//	KPV15du	: BOOL;
END_VAR
(* global variable list tmr *)
{attribute 'qualified_only' := ''}
{attribute 'symbol' := 'none'}
VAR_GLOBAL
	///Unlock
	//Unlock: Ttonp := (pt := TIME#3s0ms);
	crsPmStarter_20	: TON := ( PT := TIME#20S0MS );	// 20	
//	crsNIgnition_10: TON := (pt := TIME#0S0MS);	// 10	
//	crsNBoost_10: TON := (pt := TIME#0S0MS);	// 10
	KPV234_wOpen	: TON := ( PT := TIME#10S0MS );	// 10
	KPV15_wOpen		: TON := ( PT := TIME#10S0MS );	// 10
	KPV15_nOpen		: TON := ( PT := TIME#10S0MS );	// 10
	// задержка выключения насосов после останова
	PNU_S_Off		: TON := ( PT := TIME#5M );	// 30 minutes // 5 minutes 14_07_2025
	// задержка отключения насосов при подкачке масла Н на этапе прогрева или охлаждения двигателя
	PNU_S_pumpH		: TOF := ( PT := TIME#1M );	// 1 minutes
END_VAR
(* global variable list acpar_handler *)
{attribute 'qualified_only' := ''}
VAR_GLOBAL
	handler: TAcparHandler;
END_VAR
(* global variable list FuelReg *)
{region INFO}
(*
Назначение: Числовые настройки
Автор     : Дергаев
Дата      : 12.05.2025 16:11:36
Версия    : 00.01.00
*)
{endregion}
{attribute 'qualified_only'}
{attribute 'symbol' := 'none'}
VAR_GLOBAL
{attribute 'symbol' := 'readwrite'}
  {attribute 'export' := '("archive":"True","communication":("cycle":"base"),"name":"Верхнее ограничение Nтк","units": "об/мин","digit": "0","limit": ("low": "0.0","high": "9000.0"))'}
  limValUpNvd  : Ttunpar := (value := REAL#8350.0, set_value := REAL#8350.0, enable_valueLimit := TRUE, lolim := REAL#0.0, hilim := REAL#9000.0, enable_direct_update := TRUE); 
{attribute 'symbol' := 'readwrite'}
  {attribute 'export' := '("archive":"True","communication":("cycle":"base"),"name":"Верхнее ограничение Nст","units": "об/мин","digit": "0","limit": ("low": "0.0","high": "9000.0"))'}
  limValUpNst  : Ttunpar := (value := REAL#8500.0, set_value := REAL#8500.0, enable_valueLimit := TRUE, lolim := REAL#0.0, hilim := REAL#9000.0, enable_direct_update := TRUE); 
{attribute 'symbol' := 'readwrite'}
  {attribute 'export' := '("archive":"True","communication":("cycle":"base"),"name":"Верхнее ограничение Тст","units": "°C","digit": "0","limit": ("low": "0.0","high": "800.0"))'}
  limValUpTst  : Ttunpar := (value := REAL#650.0, set_value := REAL#650.0, enable_valueLimit := TRUE, lolim := REAL#0.0, hilim := REAL#800.0, enable_direct_update := TRUE); 
{attribute 'symbol' := 'readwrite'}
  {attribute 'export' := '("archive":"True","communication":("cycle":"base"),"name":"Верх. огр. Тст на пуске","units": "°С","digit": "0","limit": ("low": "0.0","high": "800.0"))'}
  limValUpTstStart : Ttunpar := (value := REAL#680.0, set_value := REAL#680.0, enable_valueLimit := TRUE, lolim := REAL#0.0, hilim := REAL#800.0, enable_direct_update := TRUE); 
{attribute 'symbol' := 'readwrite'}
  {attribute 'export' := '("archive":"True","communication":("cycle":"base"),"name":"Верхнее ограничение Рк","units": "МПа","digit": "2","limit": ("low": "0.0","high": "2.0"))'}
  limValUpPk  : Ttunpar := (value := REAL#1.4, set_value := REAL#1.4, enable_valueLimit := TRUE, lolim := REAL#0.0, hilim := REAL#2.0, enable_direct_update := TRUE); 
{attribute 'symbol' := 'readwrite'}
  {attribute 'export' := '("archive":"True","communication":("cycle":"base"),"name":"Рег. Верхнее ограничение Nтк","units": "об/мин","digit": "0","limit": ("low": "-500.0","high": "500.0"))'}
  RegLimValUpNvd  : Ttunpar := (value := REAL#0.0, set_value := REAL#0.0, enable_valueLimit := TRUE, lolim := REAL#-500.0, hilim := REAL#500.0, enable_direct_update := TRUE); 
{attribute 'symbol' := 'readwrite'}
  {attribute 'export' := '("archive":"True","communication":("cycle":"base"),"name":"Рег. Нижнее ограничение Nтк","units": "об/мин","digit": "0","limit": ("low": "-500.0","high": "500.0"))'}
  RegLimValDnNvd  : Ttunpar := (value := REAL#300.0, set_value := REAL#300.0, enable_valueLimit := TRUE, lolim := REAL#-500.0, hilim := REAL#500.0, enable_direct_update := TRUE); 
{attribute 'symbol' := 'readwrite'}
  {attribute 'export' := '("archive":"True","communication":("cycle":"base"),"name":"Рег. Верхнее ограничение Nст","units": "об/мин","digit": "0","limit": ("low": "-500.0","high": "500.0"))'}
  RegLimValUpNst  : Ttunpar := (value := REAL#0.0, set_value := REAL#0.0, enable_valueLimit := TRUE, lolim := REAL#-500.0, hilim := REAL#500.0, enable_direct_update := TRUE); 
{attribute 'symbol' := 'readwrite'}
  {attribute 'export' := '("archive":"True","communication":("cycle":"base"),"name":"Рег. Верхнее ограничение Тст","units": "°C","digit": "0","limit": ("low": "-200.0","high": "200.0"))'}
  RegLimValUpTst  : Ttunpar := (value := REAL#0.0, set_value := REAL#0.0, enable_valueLimit := TRUE, lolim := REAL#-200.0, hilim := REAL#200.0, enable_direct_update := TRUE); 
{attribute 'symbol' := 'readwrite'}
  {attribute 'export' := '("archive":"True","communication":("cycle":"base"),"name":"Рег. Верх. огр. Тст на пуске","units": "°С","digit": "0","limit": ("low": "-200.0","high": "200.0"))'}
  RegLimValUpTstStart : Ttunpar := (value := REAL#0.0, set_value := REAL#0.0, enable_valueLimit := TRUE, lolim := REAL#-200.0, hilim := REAL#200.0, enable_direct_update := TRUE); 
{attribute 'symbol' := 'readwrite'}
  {attribute 'export' := '("archive":"True","communication":("cycle":"base"),"name":"Рег. Верхнее ограничение Рк","units": "МПа","digit": "2","limit": ("low": "-0.5","high": "0.5"))'}
  RegLimValUpPk  : Ttunpar := (value := REAL#0.0, set_value := REAL#0.0, enable_valueLimit := TRUE, lolim := REAL#-0.5, hilim := REAL#0.5, enable_direct_update := TRUE); 
{attribute 'symbol' := 'readwrite'}
  {attribute 'export' := '("archive":"True","communication":("cycle":"base"),"name":"Ступенька на розжиг ","units": "кг/ч","digit": "0","limit": ("low": "0.0","high": "1000.0"))'}
  ignitionStep  : Ttunpar := (value := REAL#100.0, set_value := REAL#100.0, enable_valueLimit := TRUE, lolim := REAL#0.0, hilim := REAL#1000.0, enable_direct_update := TRUE); 
{attribute 'symbol' := 'readwrite'}
  {attribute 'export' := '("archive":"True","communication":("cycle":"base"),"name":"Пауза на первой ступеньке ","units": "с","digit": "0","limit": ("low": "0.0","high": "60.0"))'}
  ignitionDelay  : Ttunpar := (value := REAL#3.0, set_value := REAL#3.0, enable_valueLimit := TRUE, lolim := REAL#0.0, hilim := REAL#60.0, enable_direct_update := TRUE); 
{attribute 'symbol' := 'readwrite'}
  {attribute 'export' := '("archive":"True","communication":("cycle":"base"),"name":"Макс. длительность розжига ","units": "с","digit": "0","limit": ("low": "0.0","high": "60.0"))'}
  ignitionMaxTime  : Ttunpar := (value := REAL#10.0, set_value := REAL#10.0, enable_valueLimit := TRUE, lolim := REAL#0.0, hilim := REAL#60.0, enable_direct_update := TRUE); 
{attribute 'symbol' := 'readwrite'}
  {attribute 'export' := '("archive":"True","communication":("cycle":"base"),"name":"Макс. Gт на розжиге","units": "кг/ч","digit": "0","limit": ("low": "0.0","high": "1000.0"))'}
  ignitionMaxVal  : Ttunpar := (value := REAL#250.0, set_value := REAL#250.0, enable_valueLimit := TRUE, lolim := REAL#0.0, hilim := REAL#1000.0, enable_direct_update := TRUE); 
{attribute 'symbol' := 'readwrite'}
  {attribute 'export' := '("archive":"True","communication":("cycle":"base"),"name":"Темп программного разгона","units": "[кг/ч]/c","digit": "0","limit": ("low": "0.0","high": "1000.0"))'}
  rateOnProg  : Ttunpar := (value := REAL#30.0, set_value := REAL#30.0, enable_valueLimit := TRUE, lolim := REAL#0.0, hilim := REAL#1000.0, enable_direct_update := TRUE); 
{attribute 'symbol' := 'readwrite'}
  {attribute 'export' := '("archive":"True","communication":("cycle":"base"),"name":"Ступенька при прог. разгоне ","units": "кг/ч","digit": "0","limit": ("low": "0.0","high": "1000.0"))'}
  stepOnProg  : Ttunpar := (value := REAL#0.0, set_value := REAL#0.0, enable_valueLimit := TRUE, lolim := REAL#0.0, hilim := REAL#1000.0, enable_direct_update := TRUE); 
{attribute 'symbol' := 'readwrite'}
  {attribute 'export' := '("archive":"True","communication":("cycle":"base"),"name":"T1 регулирования Nтк","units": "с","digit": "2","limit": ("low": "0.0","high": "10.0"))'}
  tau1vd  : Ttunpar := (value := REAL#0.5, set_value := REAL#0.5, enable_valueLimit := TRUE, lolim := REAL#0.0, hilim := REAL#10.0, enable_direct_update := TRUE); 
{attribute 'symbol' := 'readwrite'}
  {attribute 'export' := '("archive":"True","communication":("cycle":"base"),"name":"T2 регулирования Nтк","units": "с","digit": "2","limit": ("low": "0.0","high": "10.0"))'}
  tau2vd  : Ttunpar := (value := REAL#0.1, set_value := REAL#0.1, enable_valueLimit := TRUE, lolim := REAL#0.0, hilim := REAL#10.0, enable_direct_update := TRUE); 
{attribute 'symbol' := 'readwrite'}
  {attribute 'export' := '("archive":"True","communication":("cycle":"base"),"name":"T1 регулирования Nст","units": "с","digit": "2","limit": ("low": "0.0","high": "10.0"))'}
  tau1st  : Ttunpar := (value := REAL#0.5, set_value := REAL#0.5, enable_valueLimit := TRUE, lolim := REAL#0.0, hilim := REAL#10.0, enable_direct_update := TRUE); 
{attribute 'symbol' := 'readwrite'}
  {attribute 'export' := '("archive":"True","communication":("cycle":"base"),"name":"Т2 регулирования Nст","units": "с","digit": "2","limit": ("low": "0.0","high": "10.0"))'}
  tau2st : Ttunpar := (value := REAL#0.1, set_value := REAL#0.1, enable_valueLimit := TRUE, lolim := REAL#0.0, hilim := REAL#10.0, enable_direct_update := TRUE); 
{attribute 'symbol' := 'readwrite'}
  {attribute 'export' := '("archive":"True","communication":("cycle":"base"),"name":"Т1 регулирования Тст","units": "с","digit": "2","limit": ("low": "0.0","high": "10.0"))'}
  tau1Tst  : Ttunpar := (value := REAL#0.5, set_value := REAL#0.5, enable_valueLimit := TRUE, lolim := REAL#0.0, hilim := REAL#10.0, enable_direct_update := TRUE); 
{attribute 'symbol' := 'readwrite'}
  {attribute 'export' := '("archive":"True","communication":("cycle":"base"),"name":"Т2 регулирования Тст","units": "с","digit": "2","limit": ("low": "0.0","high": "10.0"))'}
  tau2Tst  : Ttunpar := (value := REAL#0.1, set_value := REAL#0.1, enable_valueLimit := TRUE, lolim := REAL#0.0, hilim := REAL#10.0, enable_direct_update := TRUE); 
{attribute 'symbol' := 'readwrite'}
  {attribute 'export' := '("archive":"True","communication":("cycle":"base"),"name":"Т1 регулирования Рк","units": "с","digit": "2","limit": ("low": "0.0","high": "10.0"))'}
  tau1Pk  : Ttunpar := (value := REAL#0.5, set_value := REAL#0.5, enable_valueLimit := TRUE, lolim := REAL#0.0, hilim := REAL#10.0, enable_direct_update := TRUE); 
{attribute 'symbol' := 'readwrite'}
  {attribute 'export' := '("archive":"True","communication":("cycle":"base"),"name":"Т2 регулирования Рк","units": "с","digit": "2","limit": ("low": "0.0","high": "10.0"))'}
  tau2Pk  : Ttunpar := (value := REAL#0.1, set_value := REAL#0.1, enable_valueLimit := TRUE, lolim := REAL#0.0, hilim := REAL#10.0, enable_direct_update := TRUE); 
{attribute 'symbol' := 'readwrite'}
  {attribute 'export' := '("archive":"True","communication":("cycle":"base"),"name":"DZ регулирования Nтк","units": "об/мин","digit": "1","limit": ("low": "0.0","high": "100.0"))'}
  dzVd  : Ttunpar := (value := REAL#2.0, set_value := REAL#2.0, enable_valueLimit := TRUE, lolim := REAL#0.0, hilim := REAL#100.0, enable_direct_update := TRUE); 
{attribute 'symbol' := 'readwrite'}
  {attribute 'export' := '("archive":"True","communication":("cycle":"base"),"name":"DZ регулирования Nст","units": "об/мин","digit": "1","limit": ("low": "0.0","high": "100.0"))'}
  dzSt  : Ttunpar := (value := REAL#2.0, set_value := REAL#2.0, enable_valueLimit := TRUE, lolim := REAL#0.0, hilim := REAL#100.0, enable_direct_update := TRUE); 
{attribute 'symbol' := 'readwrite'}
  {attribute 'export' := '("archive":"True","communication":("cycle":"base"),"name":"DZ регулирования Тст","units": "°С","digit": "1","limit": ("low": "0.0","high": "100.0"))'}
  dzTst  : Ttunpar := (value := REAL#1.0, set_value := REAL#1.0, enable_valueLimit := TRUE, lolim := REAL#0.0, hilim := REAL#100.0, enable_direct_update := TRUE); 
{attribute 'symbol' := 'readwrite'}
  {attribute 'export' := '("archive":"True","communication":("cycle":"base"),"name":"DZ регулирования Рк","units": "МПа","digit": "2","limit": ("low": "0.0","high": "0.2"))'}
  dzPk  : Ttunpar := (value := REAL#0.01, set_value := REAL#0.01, enable_valueLimit := TRUE, lolim := REAL#0.0, hilim := REAL#0.2, enable_direct_update := TRUE); 
{attribute 'symbol' := 'readwrite'}
  {attribute 'export' := '("archive":"True","communication":("cycle":"base"),"name":"К рабочего регулятора Nтк","units": "","digit": "2","limit": ("low": "0.0","high": "50.0"))'}
  kRVd  : Ttunpar := (value := REAL#0.0001, set_value := REAL#0.0001, enable_valueLimit := TRUE, lolim := REAL#0.0, hilim := REAL#50.0, enable_direct_update := TRUE); 
{attribute 'symbol' := 'readwrite'}
  {attribute 'export' := '("archive":"True","communication":("cycle":"base"),"name":"К верхнего ограничителя Nтк","units": "","digit": "2","limit": ("low": "0.0","high": "50.0"))'}
  kLupVd  : Ttunpar := (value := REAL#0.1, set_value := REAL#0.1, enable_valueLimit := TRUE, lolim := REAL#0.0, hilim := REAL#50.0, enable_direct_update := TRUE); 
{attribute 'symbol' := 'readwrite'}
  {attribute 'export' := '("archive":"True","communication":("cycle":"base"),"name":"К нижнего ограничителя Nтк","units": "","digit": "2","limit": ("low": "0.0","high": "50.0"))'}
  kLdnVd  : Ttunpar := (value := REAL#0.1, set_value := REAL#0.1, enable_valueLimit := TRUE, lolim := REAL#0.0, hilim := REAL#50.0, enable_direct_update := TRUE); 
{attribute 'symbol' := 'readwrite'}
  {attribute 'export' := '("archive":"True","communication":("cycle":"base"),"name":"К рабочего регулятора Nст","units": "","digit": "2","limit": ("low": "0.0","high": "50.0"))'}
  kRst  : Ttunpar := (value := REAL#0.0001, set_value := REAL#0.0001, enable_valueLimit := TRUE, lolim := REAL#0.0, hilim := REAL#50.0, enable_direct_update := TRUE); 
{attribute 'symbol' := 'readwrite'}
  {attribute 'export' := '("archive":"True","communication":("cycle":"base"),"name":"К верхнего ограничителя Nст","units": "","digit": "2","limit": ("low": "0.0","high": "50.0"))'}
  kLupST  : Ttunpar := (value := REAL#0.1, set_value := REAL#0.1, enable_valueLimit := TRUE, lolim := REAL#0.0, hilim := REAL#50.0, enable_direct_update := TRUE); 
{attribute 'symbol' := 'readwrite'}
  {attribute 'export' := '("archive":"True","communication":("cycle":"base"),"name":"К верхнего ограничителя Тст","units": "","digit": "2","limit": ("low": "0.0","high": "50.0"))'}
  kLupTst  : Ttunpar := (value := REAL#0.1, set_value := REAL#0.1, enable_valueLimit := TRUE, lolim := REAL#0.0, hilim := REAL#50.0, enable_direct_update := TRUE); 
{attribute 'symbol' := 'readwrite'}
  {attribute 'export' := '("archive":"True","communication":("cycle":"base"),"name":"К верхнего ограничителя Рк","units": "","digit": "2","limit": ("low": "0.0","high": "50.0"))'}
  kLupPk  : Ttunpar := (value := REAL#0.1, set_value := REAL#0.1, enable_valueLimit := TRUE, lolim := REAL#0.0, hilim := REAL#50.0, enable_direct_update := TRUE); 
{attribute 'symbol' := 'readwrite'}
  {attribute 'export' := '("archive":"True","communication":("cycle":"base"),"name":"К коррекции Nтк","units": "[об/мин]/[кг/ч]","digit": "4","limit": ("low": "0.0","high": "50.0"))'}
   kCorrNvd : Ttunpar := (value := REAL#4.0, set_value := REAL#4.0, enable_valueLimit := TRUE, lolim := REAL#0.0, hilim := REAL#50.0, enable_direct_update := TRUE); 
{attribute 'symbol' := 'readwrite'}
  {attribute 'export' := '("archive":"True","communication":("cycle":"base"),"name":"К коррекции Nст","units": "[об/мин]/[кг/ч]","digit": "4","limit": ("low": "0.0","high": "50.0"))'}
   kCorrNst : Ttunpar := (value := REAL#4.0, set_value := REAL#4.0, enable_valueLimit := TRUE, lolim := REAL#0.0, hilim := REAL#50.0, enable_direct_update := TRUE); 
{attribute 'symbol' := 'readwrite'}
  {attribute 'export' := '("archive":"True","communication":("cycle":"base"),"name":"К коррекции Tст","units": "°С/[кг/ч]","digit": "1","limit": ("low": "0.0","high": "50.0"))'}
   kCorrTst : Ttunpar := (value := REAL#0.3, set_value := REAL#0.3, enable_valueLimit := TRUE, lolim := REAL#0.0, hilim := REAL#50.0, enable_direct_update := TRUE); 
{attribute 'symbol' := 'readwrite'}
  {attribute 'export' := '("archive":"True","communication":("cycle":"base"),"name":"К коррекции Рк","units": "МПа/[кг/ч]","digit": "1","limit": ("low": "0.0","high": "50.0"))'}
   kCorrPk  : Ttunpar := (value := REAL#0.0005, set_value := REAL#0.0005, enable_valueLimit := TRUE, lolim := REAL#0.0, hilim := REAL#50.0, enable_direct_update := TRUE); 
{attribute 'symbol' := 'readwrite'}
  {attribute 'export' := '("archive":"True","communication":("cycle":"base"),"name":"Обороты вкл. рег. по Nтк","units": "об/мин","digit": "0","limit": ("low": "0.0","high": "8000.0"))'}
  setNvdRegOn  : Ttunpar := (value := REAL#6300.0, set_value := REAL#6300.0, enable_valueLimit := TRUE, lolim := REAL#0.0, hilim := REAL#8000.0, enable_direct_update := TRUE); 
{attribute 'symbol' := 'readwrite'}
  {attribute 'export' := '("archive":"True","communication":("cycle":"base"),"name":"Обороты выключения стартера","units": "об/мин","digit": "0","limit": ("low": "0.0","high": "8000.0"))'}
  setNvdStarterOff  : Ttunpar := (value := REAL#4500.0, set_value := REAL#4500.0, enable_valueLimit := TRUE, lolim := REAL#0.0, hilim := REAL#8000.0, enable_direct_update := TRUE); 
{attribute 'symbol' := 'readwrite'}
  {attribute 'export' := '("archive":"True","communication":("cycle":"base"),"name":"Обороты прогрева","units": "об/мин","digit": "0","limit": ("low": "0.0","high": "8000.0"))'}
  setNvdHeat  : Ttunpar := (value := REAL#6800.0, set_value := REAL#6800.0, enable_valueLimit := TRUE, lolim := REAL#0.0, hilim := REAL#8000.0, enable_direct_update := TRUE); 
{attribute 'symbol' := 'readwrite'}
  {attribute 'export' := '("archive":"True","communication":("cycle":"base"),"name":"Время прогрева","units": "с","digit": "0","limit": ("low": "0.0","high": "500.0"))'}
  setHeatTime  : Ttunpar := (value := REAL#300.0, set_value := REAL#300.0, enable_valueLimit := TRUE, lolim := REAL#0.0, hilim := REAL#500.0, enable_direct_update := TRUE); 
{attribute 'symbol' := 'readwrite'}
  {attribute 'export' := '("archive":"True","communication":("cycle":"base"),"name":"Обороты охлаждения","units": "об/мин","digit": "0","limit": ("low": "0.0","high": "8000.0"))'}
  setNvdCool  : Ttunpar := (value := REAL#6700.0, set_value := REAL#6700.0, enable_valueLimit := TRUE, lolim := REAL#0.0, hilim := REAL#8000.0, enable_direct_update := TRUE); 
{attribute 'symbol' := 'readwrite'}
  {attribute 'export' := '("archive":"True","communication":("cycle":"base"),"name":"Время охлаждения","units": "с","digit": "0","limit": ("low": "0.0","high": "500.0"))'}
  setCoolTime  : Ttunpar := (value := REAL#300.0, set_value := REAL#300.0, enable_valueLimit := TRUE, lolim := REAL#0.0, hilim := REAL#500.0, enable_direct_update := TRUE); 
{attribute 'symbol' := 'readwrite'}
  {attribute 'export' := '("archive":"True","communication":("cycle":"base"),"name":"Ступенька Т на пуске","units": "°С","digit": "0","limit": ("low": "0.0","high": "500.0"))'}
  setDTign  : Ttunpar := (value := REAL#100.0, set_value := REAL#100.0, enable_valueLimit := TRUE, lolim := REAL#0.0, hilim := REAL#500.0, enable_direct_update := TRUE); 
{attribute 'symbol' := 'readwrite'}
  {attribute 'export' := '("archive":"True","communication":("cycle":"base"),"name":"dNтк до верх. границы - сигн.","units": "об/мин","digit": "0","limit": ("low": "0.0","high": "100.0"))'}
  dNvdUpLim : Ttunpar := (value := REAL#20.0, set_value := REAL#20.0, enable_valueLimit := TRUE, lolim := REAL#0.0, hilim := REAL#100.0, enable_direct_update := TRUE); 
{attribute 'symbol' := 'readwrite'}
  {attribute 'export' := '("archive":"True","communication":("cycle":"base"),"name":"dNтк до нижн. границы - сигн.","units": "об/мин","digit": "0","limit": ("low": "0.0","high": "100.0"))'}
  dNvdDnLim : Ttunpar := (value := REAL#20.0, set_value := REAL#20.0, enable_valueLimit := TRUE, lolim := REAL#0.0, hilim := REAL#100.0, enable_direct_update := TRUE); 
{attribute 'symbol' := 'readwrite'}
  {attribute 'export' := '("archive":"True","communication":("cycle":"base"),"name":"dNст до верх. границы - сигн.","units": "об/мин","digit": "0","limit": ("low": "0.0","high": "100.0"))'}
  dNstUpLim : Ttunpar := (value := REAL#20.0, set_value := REAL#20.0, enable_valueLimit := TRUE, lolim := REAL#0.0, hilim := REAL#100.0, enable_direct_update := TRUE); 
{attribute 'symbol' := 'readwrite'}
  {attribute 'export' := '("archive":"True","communication":("cycle":"base"),"name":"dТст до верх. границы - сигн.","units": "°С","digit": "0","limit": ("low": "0.0","high": "100.0"))'}
  dTstUpLim : Ttunpar := (value := REAL#10.0, set_value := REAL#10.0, enable_valueLimit := TRUE, lolim := REAL#0.0, hilim := REAL#100.0, enable_direct_update := TRUE); 
{attribute 'symbol' := 'readwrite'}
  {attribute 'export' := '("archive":"True","communication":("cycle":"base"),"name":"dPk до верх. границы - сигн.","units": "МПа","digit": "2","limit": ("low": "0.0","high": "0.5"))'}
  dPkUpLim : Ttunpar := (value := REAL#0.1, set_value := REAL#0.1, enable_valueLimit := TRUE, lolim := REAL#0.0, hilim := REAL#0.5, enable_direct_update := TRUE); 
{attribute 'symbol' := 'readwrite'}
  {attribute 'export' := '("archive":"True","communication":("cycle":"base"),"name":"Мин. Т при работе - горение","units": "°С","digit": "0","limit": ("low": "0.0","high": "700.0"))'}
  lowTonWork : Ttunpar := (value := REAL#250.0, set_value := REAL#250.0, enable_valueLimit := TRUE, lolim := REAL#0.0, hilim := REAL#700.0, enable_direct_update := TRUE); 
{attribute 'symbol' := 'readwrite'}
  {attribute 'export' := '("archive":"True","communication":("cycle":"base"),"name":"Задержка контроля Мин.Т","units": "с","digit": "0","limit": ("low": "0.0","high": "100.0"))'}
  delayLowTonWork : Ttunpar := (value := REAL#10.0, set_value := REAL#10.0, enable_valueLimit := TRUE, lolim := REAL#0.0, hilim := REAL#100.0, enable_direct_update := TRUE); 
{attribute 'symbol' := 'readwrite'}
  {attribute 'export' := '("archive":"True","communication":("cycle":"base"),"name":"Темп разгона на регуляторе","units": "(об/мин)/c","digit": "0","limit": ("low": "0.0","high": "200.0"))'}
  rateOnReg  : Ttunpar := (value := REAL#50.0, set_value := REAL#50.0, enable_valueLimit := TRUE, lolim := REAL#0.0, hilim := REAL#200.0, enable_direct_update := TRUE); 
  // Обратная зависимость расхода топлива от степени открытия топливного клапана
  gTtoDoz : Tlinear :=
  (
    nPoint :=  17,
    point :=
    [
      (x := REAL#0.0, y := REAL#0.0),
      (x := REAL#117.0, y := REAL#6.25),
      (x := REAL#330.0, y := REAL#12.5),
      (x := REAL#555.0, y := REAL#18.75),
      (x := REAL#757.0, y := REAL#25.0),
      (x := REAL#995.0, y := REAL#31.25),
      (x := REAL#1250.0, y := REAL#37.5),
      (x := REAL#1522.0, y := REAL#43.75),
      (x := REAL#1806.0, y := REAL#50.0),
      (x := REAL#2107.0, y := REAL#56.25),
      (x := REAL#2430.0, y := REAL#62.5),
      (x := REAL#2772.0, y := REAL#68.75),
      (x := REAL#3135.0, y := REAL#75.0),
      (x := REAL#3527.0, y := REAL#81.25),
      (x := REAL#3948.0, y := REAL#87.5),
      (x := REAL#4412.0, y := REAL#93.75),
      (x := REAL#4920.0, y := REAL#100.0)
    ]
  );

  {attribute 'symbol' := 'read'}
  fReg : TRegNK12ST;
END_VAR
(* global variable list PRU *)
{attribute 'symbol' := 'read'}
{attribute 'qualified_only' := ''}
VAR_GLOBAL
	/// связь с ПРУ
	/// FALSE - отсутствие связи
	Link: BOOL;
END_VAR
(* global variable list AVOM *)
{attribute 'qualified_only' := ''}
VAR_GLOBAL
	AVOM: TAVOM;
END_VAR
(* global variable list lmt *)
{region INFO}
(*
 Назначение: Признаки срабатывания ограничительных сигнализаций
 Автор:  /Andrey/ 24.06.2025 16:50:31
 Версия: v00.00.22
 Проект: KA107__GPA2
*)
{endregion}
{attribute 'qualified_only'}
{attribute 'symbol' := 'read'}
VAR_GLOBAL
	{attribute 'symbol' := 'none'}
	common : Talarm; //Общий сигнал для VAR_STAT

END_VAR
(* global variable list BZA *)
{attribute 'symbol' := 'none'}
VAR_GLOBAL CONSTANT
	/// Уставка + доп. коэффициент
	Nst_SetUp: REAL := 3500;//2000;
	/// Уставка + доп. коэффициент
	Ntk_SetUp: REAL := 6000;//2000;
END_VAR
(* global variable list ACS *)
{attribute 'qualified_only'}
VAR_GLOBAL
	ACS			: TAutoCheckShield;
	startACS	: BOOL;		// Пуск проверки
END_VAR
(* global variable list IEC104 *)
{region INFO}
(*
 Назначение: Используется для объявления переменных, предназначенных для передачи по МЭК-104
 Автор:      /Andrey/ 16.07.2025 17:15:07
*)
{endregion}
{attribute 'qualified_only'}
{attribute 'symbol' := 'none'}
VAR_GLOBAL
	{attribute 'export' := 'an:[GVL.mde_hmi] af:[.number]'}
	GVL_mde_hmi_number : PsIEC60870.m_it_tb_1_fb; //Режим/Тип:int4/Адрес:1
	{attribute 'export' := 'an:[test.Saw_Slow] af:[.value]'}
	test_Saw_Slow_value : PsIEC60870.m_me_tf_1_fb; //Тест: пила, базовый цикл/Тип:REAL/Адрес:2
	{attribute 'export' := 'an:[test.Saw_Fast] af:[.value]'}
	test_Saw_Fast_value : PsIEC60870.m_me_tf_1_fb; //Тест: пила, быстрый цикл/Тип:REAL/Адрес:3
	{attribute 'export' := 'an:[test.Sin_Slow] af:[.value]'}
	test_Sin_Slow_value : PsIEC60870.m_me_tf_1_fb; //Тест: синус, базовый цикл/Тип:REAL/Адрес:4
	{attribute 'export' := 'an:[aipar.NTK_1] af:[.in_value]'}
	aipar_NTK_1_in_value : PsIEC60870.m_me_tf_1_fb; //Частота вращения ротора ТК (1)/Тип:REAL/Адрес:5
	{attribute 'export' := 'an:[aipar.NTK_2] af:[.in_value]'}
	aipar_NTK_2_in_value : PsIEC60870.m_me_tf_1_fb; //Частота вращения ротора ТК (2)/Тип:REAL/Адрес:6
	{attribute 'export' := 'an:[aipar.NST_1] af:[.in_value]'}
	aipar_NST_1_in_value : PsIEC60870.m_me_tf_1_fb; //Частота вращения ротора СТ (1)/Тип:REAL/Адрес:7
	{attribute 'export' := 'an:[aipar.NST_2] af:[.in_value]'}
	aipar_NST_2_in_value : PsIEC60870.m_me_tf_1_fb; //Частота вращения ротора СТ (2)/Тип:REAL/Адрес:8
	{attribute 'export' := 'an:[aipar.DG_Pos] af:[.in_value]'}
	aipar_DG_Pos_in_value : PsIEC60870.m_me_tf_1_fb; //Положение дозирующей иглы ДУС/Тип:REAL/Адрес:9
	{attribute 'export' := 'an:[aipar.Pa_out14] af:[.in_value]'}
	aipar_Pa_out14_in_value : PsIEC60870.m_me_tf_1_fb; //Давление воздуха за 14-й ступенью осевого компрессора/Тип:REAL/Адрес:10
	{attribute 'export' := 'an:[aipar.dP_conf] af:[.in_value]'}
	aipar_dP_conf_in_value : PsIEC60870.m_me_tf_1_fb; //dP на конфузоре/Тип:REAL/Адрес:11
	{attribute 'export' := 'an:[aopar.DG_Set] af:[.value]'}
	aopar_DG_Set_value : PsIEC60870.m_me_tf_1_fb; //Управление ТРК/Тип:REAL/Адрес:12
	{attribute 'export' := 'an:[dipar.SK_off] af:[.status]'}
	dipar_SK_off_status : PsIEC60870.m_bo_tb_1_fb; //СК закрыт/Тип:uint4/Адрес:13
	{attribute 'export' := 'an:[dopar.SK_ON] af:[.status]'}
	dopar_SK_ON_status : PsIEC60870.m_bo_tb_1_fb; //Открыть СК/Тип:uint4/Адрес:14
	{attribute 'export' := 'an:[aipar.DG_Pos_diag] af:[.in_value]'}
	aipar_DG_Pos_diag_in_value : PsIEC60870.m_me_tf_1_fb; //диаг. (Сигнал управления положением дозатора газа)/Тип:REAL/Адрес:15
	{attribute 'export' := 'an:[dopar.KPV15_ON] af:[.status]'}
	dopar_KPV15_ON_status : PsIEC60870.m_bo_tb_1_fb; //Открыть КПВ1, 5/Тип:uint4/Адрес:16
END_VAR
(* global variable list test *)
{attribute 'qualified_only'}
VAR_GLOBAL
	Saw_Slow	: TATestpar := ( sin_on := FALSE );
	Saw_Fast	: TATestpar := ( sin_on := FALSE );
	Sin_Slow	: TATestpar;
END_VAR
(* global variable list s_tunpar *)
{region INFO}
(*
Назначение: Числовые настройки
Автор     : Дергаев
Дата      : 20.03.2025 16:19:20
Версия    : 00.00.02
*)
{endregion}
{attribute 'qualified_only'}
{attribute 'symbol' := 'readwrite'}
VAR_GLOBAL
  {attribute 'symbol' := 'none'}
  {attribute 'export' := 'a n:[Задержка на снятие сигнала "Предпомпажное состояние"] u:[с] d:[1] lolim:[0] hilim:[1000]'}
  SAoffDelay : Ttunpar := (value := REAL#0.5, set_value := REAL#0.5, enable_direct_update := TRUE); 
  {attribute 'symbol' := 'none'}
  {attribute 'export' := 'a n:[Задержка на открытие АПРК при срабатывании сигнализатора помпажа] u:[с] d:[1] lolim:[0] hilim:[1000]'}
  SAopenDelay : Ttunpar := (value := REAL#0.0, set_value := REAL#0.0, enable_direct_update := TRUE); 
  {attribute 'symbol' := 'none'}
  {attribute 'export' := 'a n:[Задержка срабатывания сигнализатора помпажа] u:[с] d:[1] lolim:[0] hilim:[1000]'}
  SAdelay : Ttunpar := (value := REAL#2.0, set_value := REAL#2.0, enable_direct_update := TRUE); 
  {attribute 'symbol' := 'none'}
  {attribute 'export' := 'a n:[Задержка на блокировку подсчета числа срабатываний диагностики предпомпажного состояния] u:[с] d:[1] lolim:[0] hilim:[1000]'}
  blockDelay : Ttunpar := (value := REAL#2.0, set_value := REAL#2.0, enable_direct_update := TRUE); 
  {attribute 'symbol' := 'none'}
  {attribute 'export' := 'a n:[Задержка на сброс счетчика числа срабатываний диагностики предпомпажного состояния] u:[с] d:[1] lolim:[0] hilim:[1000]'}
  resetDelay : Ttunpar := (value := REAL#10.0, set_value := REAL#10.0, enable_direct_update := TRUE); 
  {attribute 'export' := 'a n:[Коэфф. при 2-й степ. осн. системы координат] u:[] d:[4] lolim:[-100] hilim:[100]'}
  c2Main : Ttunpar := (value := REAL#-0.4951, set_value := REAL#-0.4951, enable_direct_update := TRUE); 
  {attribute 'export' := 'a n:[Коэфф. при 1-й степ. осн. системы координат] u:[] d:[4] lolim:[-100] hilim:[100]'}
  c1Main : Ttunpar := (value := REAL#1.032, set_value := REAL#1.032, enable_direct_update := TRUE); 
  {attribute 'export' := 'a n:[Коэфф. при 0-й степ. осн. системы координат] u:[] d:[4] lolim:[-100] hilim:[100]'}
  c0Main : Ttunpar := (value := REAL#1.7225, set_value := REAL#1.7225, enable_direct_update := TRUE); 
  {attribute 'export' := 'a n:[Коэфф. при 2-й степ. 1-й рез. системы координат] u:[] d:[4] lolim:[-100] hilim:[100]'}
  c2Res1 : Ttunpar := (value := REAL#-0.3076, set_value := REAL#-0.3076, enable_direct_update := TRUE); 
  {attribute 'export' := 'a n:[Коэфф. при 1-й степ. 1-й рез. системы координат] u:[] d:[4] lolim:[-100] hilim:[100]'}
  c1Res1 : Ttunpar := (value := REAL#1.0322, set_value := REAL#1.0322, enable_direct_update := TRUE); 
  {attribute 'export' := 'a n:[Коэфф. при 0-й степ. 1-й рез. системы координат] u:[] d:[4] lolim:[-100] hilim:[100]'}
  c0Res1 : Ttunpar := (value := REAL#1.4, set_value := REAL#1.4, enable_direct_update := TRUE); 
  {attribute 'export' := 'a n:[Коэфф. при 2-й степ. 2-й рез. системы координат] u:[] d:[4] lolim:[-100] hilim:[100]'}
  c2Res2 : Ttunpar := (value := REAL#1.5895, set_value := REAL#1.5895, enable_direct_update := TRUE); 
  {attribute 'export' := 'a n:[Коэфф. при 1-й степ. 2-й рез. системы координат] u:[] d:[4] lolim:[-100] hilim:[100]'}
  c1Res2 : Ttunpar := (value := REAL#-1.7931, set_value := REAL#-1.7931, enable_direct_update := TRUE); 
  {attribute 'export' := 'a n:[Коэфф. при 0-й степ. 2-й рез. системы координат] u:[] d:[4] lolim:[-100] hilim:[100]'}
  c0Res2 : Ttunpar := (value := REAL#1.7433, set_value := REAL#1.7433, enable_direct_update := TRUE); 
  {attribute 'export' := 'a n:[Мин. помпажный запас] u:[%] d:[1] lolim:[0] hilim:[100]'}
  minSR : Ttunpar := (value := REAL#10.0, set_value := REAL#10.0, enable_direct_update := TRUE); 
  {attribute 'export' := 'a n:[Макс. давление на выходе Н] u:[МПа] d:[2] lolim:[0] hilim:[32]'}
  maxPout  : Ttunpar := (value := REAL#7.5, set_value := REAL#7.5, enable_direct_update := TRUE); 
  {attribute 'export' := 'a n:[Макс. степень сжатия] u:[] d:[2] lolim:[0] hilim:[3]'}
  maxPR  : Ttunpar := (value := REAL#1.27, set_value := REAL#1.27, enable_direct_update := TRUE); 
  {attribute 'export' := 'a n:[Коэффициент конфузора] u:[] d:[2] lolim:[0] hilim:[1000]'}
  Kconf : Ttunpar := (value := REAL#44.18806572, set_value := REAL#44.18806572, enable_direct_update := TRUE); 
  {attribute 'export' := 'a n:[Номинальная N СТ] u:[об/мин] d:[0] lolim:[0] hilim:[10000]'}
  nNorm  : Ttunpar := (value := REAL#8200.0, set_value := REAL#8200.0, enable_direct_update := TRUE); 
  {attribute 'export' := 'a n:[Макс. ск. падения dP на конфузоре] u:[кПа/с] d:[1] lolim:[0] hilim:[1000]'}
  maxRateDPconf  : Ttunpar := (value := REAL#40.0, set_value := REAL#40.0, enable_direct_update := TRUE); 
  {attribute 'export' := 'a n:[Макс. ск. нарастания N СТ] u:[[об/мин]/с] d:[1] lolim:[0] hilim:[1000]'}
  maxRateNst  : Ttunpar := (value := REAL#1000.0, set_value := REAL#1000.0, enable_direct_update := TRUE); 
  {attribute 'export' := 'a n:[Макс. ск. падения помпажного запаса] u:[%/с] d:[1] lolim:[0] hilim:[100]'}
  maxRateSR : Ttunpar := (value := REAL#10.0, set_value := REAL#10.0, enable_direct_update := TRUE); 
  {attribute 'export' := 'a n:[Макс. ск. падения помпажного запаса К->М] u:[%/с] d:[1] lolim:[0] hilim:[100]'}
  maxRateSR_KM : Ttunpar := (value := REAL#20.0, set_value := REAL#20.0, enable_direct_update := TRUE); 
  {attribute 'symbol' := 'read'}
  ASprot : TASProtector;
END_VAR
(* global variable list GVL_HAND_DIAGN *)
{attribute 'symbol' := 'readwrite'}
VAR_GLOBAL
	MODULE_UPD1_A1_DI1: PsDiagn.MODULE_DI_16_012;
	MODULE_UPD1_A1_DI2: PsDiagn.MODULE_DI_16_012;
	MODULE_UPD1_A1_DI3: PsDiagn.MODULE_DI_16_012;
END_VAR
(* global variable list KPV *)
{attribute 'symbol' := 'none'}
VAR_GLOBAL CONSTANT
		// Обороты ТК, при которых происходят указанные действия
	Ntk_KPV15Close	: REAL := 7700;
	Ntk_KPV15Open	: REAL := 7600;
	Ntk_KPVClose	: REAL := 2100;
END_VAR
(* global variable list sequences *)
{region INFO}
(*
 Назначение: Используется для автоматического объявления экземпляров функциональных блоков последовательностей
 Автор:      /Разработчик/ 08.08.2025 9:04:03
 Версия:     v00.00.18
 Проект:     KA107
*)
{endregion}
{attribute 'symbol' := 'read'}
VAR_GLOBAL
{attribute 'export' := '(
    "type": "TSequence",
    "sequence": (
        "Group": "Режимные",
        "AlgGroup": "smd",
        "Name": "ХП",
        "Alg": "[HP]",
        "Items": [
            (
                "Transition": "0→1",
                "Condition": "Режим ХП",
                "AlgCondition": "[mde.HP]"
            ),
            (
                "Step": "1",
                "Commands": [
                    (
                        "Command": "Предпусковая сигнализация",
                        "AlgCommand": "[cmd_sound_On]"
                    )
                ]
            ),
            (
                "Transition": "1→2",
                "Condition": "Логическая 1",
                "AlgCondition": "[TRUE]",
                "DelayTime": "10"
            ),
            (
                "Step": "2",
                "Commands": [
                    (
                        "Command": "Пуск маслонасосов смазки и уплотнения",
                        "AlgCommand": "[cmd_PNU_S_On]"
                    )
                ]
            ),
            (
                "Transition": "2→3",
                "Condition": "dP масло-газ > 0.5 кгс/см2 и Pm > 1 кгс/см2",
                "AlgCondition": "[aipar.dPmg.value > 0.5 AND NOT dipar.Pm_N_Pn.value]"
            ),
            (
                "Step": "3",
                "Commands": [
                    (
                        "Command": "Взвод защиты по маслосистеме нагнетателя",
                        "AlgCommand": "[cmd_shPmN_On]"
                    ),
                    (
                        "Command": "Взвод защиты по перепаду \"масло-газ\"",
                        "AlgCommand": "[cmd_sh_dPmg_On]"
                    ),
                    (
                        "Command": "Открытие крана 11, закрытие крана 10",
                        "AlgCommand": "[cmd_KR11_On]",
                        "Fault": "Кран 11 не открылся, кран 10 не закрылся",
                        "AlgFault": "[am.KR11.notOn OR am.KR10.notOff]"
                    )
                ]
            ),
            (
                "Transition": "3→4",
                "Condition": "Кран 11 открылся, кран 10 закрылся",
                "AlgCondition": "[am.KR11.isOn AND am.KR10.isOff]"
            ),
            (
                "Step": "4",
                "Commands": [
                    (
                        "Command": "Проверка Nвд",
                        "AlgCommand": "[check]",
                        "Fault": "Nвд > 100 об/мин",
                        "AlgFault": "[acpar.Ntk.value > 100.0]"
                    )
                ]
            ),
            (
                "Transition": "4→5",
                "Condition": "Nвд < 100 об/мин",
                "AlgCondition": "[acpar.Ntk.value < 100.0]"
            ),
            (
                "Step": "5",
                "Commands": [
                    (
                        "Command": "Пуск воздушного стартера",
                        "AlgCommand": "[cmd_VS_On]",
                        "Fault": "Кран 13 не открылся",
                        "AlgFault": "[am.KR13.notOn]",
                        "Classifier": "P"
                    )
                ]
            ),
            (
                "Transition": "5→6",
                "Condition": "Логическая 1",
                "AlgCondition": "[TRUE]"
            ),
            (
                "Step": "6",
                "Commands": [
                    (
                        "Command": "Взвод защиты по давлению масла ВС",
                        "AlgCommand": "[cmd_sh_Pm_Starter]",
                        "Classifier": "P"
                    ),
                    (
                        "Command": "Холодная прокрутка двигателя",
                        "AlgCommand": "[cmd_HP_D]",
                        "Classifier": "P"
                    )
                ]
            ),
            (
                "Transition": "6→7",
                "Condition": "Логическая 1",
                "AlgCondition": "[TRUE]",
                "DelayTime": "120"
            ),
            (
                "Step": "7",
                "Commands": [
                    (
                        "Command": "Останов воздушного стартера",
                        "AlgCommand": "[cmd_VS_Off]",
                        "Fault": "Кран 13 не закрылся",
                        "AlgFault": "[am.KR13.notOff]"
                    )
                ]
            ),
            (
                "Transition": "7→8",
                "Condition": "Холодная прокрутка двигателя завершена",
                "AlgCondition": "[am.KR13.isOff]"
            ),
            (
                "Step": "8",
                "Commands": [
                    (
                        "Command": "Закрытие крана 11, открытие крана 10",
                        "AlgCommand": "[cmd_KR11_Off]",
                        "Fault": "Кран 11 не закрылся, кран 10 не открылся",
                        "AlgFault": "[am.KR11.notOff OR am.KR10.notOn]"
                    ),
                    (
                        "Command": "Выбег двигателя после ХП",
                        "AlgCommand": "[cmd_HP_stop_D]"
                    )
                ]
            ),
            (
                "Transition": "8→9",
                "Condition": "Nтк < 100 И Нет газа в контуре",
                "AlgCondition": "[acpar.Ntk.value < 100 AND tch.nGas_N.value]"
            ),
            (
                "Transition": "8→11",
                "Condition": "Nтк < 100 И Есть газ в контуре",
                "AlgCondition": "[acpar.Ntk.value < 100 AND tch.Gas_N.value]"
            ),
            (
                "Step": "9",
                "Commands": [
                    (
                        "Command": "Снятие защиты по маслосистеме",
                        "AlgCommand": "[cmd_shPmN_Off]"
                    ),
                    (
                        "Command": "Отключение маслонасоса уплотнения",
                        "AlgCommand": "[cmd_PNU_Off]",
                        "Fault": "Маслонасос уплотнений не выключился",
                        "AlgFault": "[am.PNU.notOff]"
                    ),
                    (
                        "Command": "Снятие защиты по перепаду \"масло-газ\"",
                        "AlgCommand": "[cmd_sh_dPmg_Off]"
                    )
                ]
            ),
            (
                "Transition": "9→10",
                "Condition": "Логическая 1",
                "AlgCondition": "[TRUE]",
                "DelayTime": "2"
            ),
            (
                "Step": "10",
                "Commands": [
                    (
                        "Command": "Отключение маслонасоса смазки",
                        "AlgCommand": "[cmd_PNS_Off]",
                        "Fault": "Маслонасос смазки не выключился",
                        "AlgFault": "[am.PNS.notOff]"
                    )
                ]
            ),
            (
                "Transition": "10→11",
                "Condition": "Логическая 1",
                "AlgCondition": "[TRUE]"
            ),
            (
                "Step": "11",
                "Commands": [
                    (
                        "Command": "Завершение",
                        "AlgCommand": "[finish]",
                        "Classifier": "P"
                    )
                ]
            ),
            (
                "Transition": "11→0",
                "Condition": "Логическая 1",
                "AlgCondition": "[TRUE]"
            ),
            (
                "Transition": "N→0",
                "Condition": "Снятие режима",
                "AlgCondition": "[NOT mde.HP]"
            )
        ]
    )
)'}
	HP : T_HP; //ХП
{attribute 'export' := '(
    "type": "TSequence",
    "sequence": (
        "Group": "Режимные",
        "AlgGroup": "smd",
        "Name": "КПК",
        "Alg": "[KPK]",
        "Items": [
            (
                "Transition": "0→1",
                "Condition": "Режим КПК",
                "AlgCondition": "[mde.KPK]"
            ),
            (
                "Step": "1",
                "Commands": [
                    (
                        "Command": "Предпусковая сигнализация",
                        "AlgCommand": "[cmd_sound_On]"
                    )
                ]
            ),
            (
                "Transition": "1→2",
                "Condition": "Логическая 1",
                "AlgCondition": "[TRUE]",
                "DelayTime": "10"
            ),
            (
                "Step": "2",
                "Commands": [
                    (
                        "Command": "Пуск маслонасосов уплотнения и смазки",
                        "AlgCommand": "[cmd_PNU_S_On]",
                        "Fault": "Маслонасос уплотнений не включился",
                        "AlgFault": "[am.PNU.notOn]"
                    )
                ]
            ),
            (
                "Transition": "2→3",
                "Condition": "dP масло-газ > 0.5 кгс/см2 и Pm > 1 кгс/см2",
                "AlgCondition": "[aipar.dPmg.value > 0.5 AND NOT dipar.Pm_N_Pn.value]"
            ),
            (
                "Step": "3",
                "Commands": [
                    (
                        "Command": "Взвод защиты по перепаду \"масло-газ\"",
                        "AlgCommand": "[cmd_sh_dPmg_On]"
                    ),
                    (
                        "Command": "Взвод защиты по маслосистеме нагнетателя",
                        "AlgCommand": "[cmd_shPmN_On]"
                    ),
                    (
                        "Command": "Запуск последовательности \"Заполнение контура компрессора\"",
                        "AlgCommand": "[cmd_filling]",
                        "Classifier": "P"
                    )
                ]
            ),
            (
                "Transition": "3→4",
                "Condition": "Подсистема \"Газовая обвязка\" запущена",
                "AlgCondition": "[subsystem.go.work]"
            ),
            (
                "Step": "4",
                "Commands": [
                    (
                        "Command": "Открытие крана 12, закрытие крана 9",
                        "AlgCommand": "[cmd_KR12_On]",
                        "Fault": "Кран 12 не открылся, кран 9 не закрылся",
                        "AlgFault": "[am.KR12.notOn OR am.KR9.notOff]"
                    )
                ]
            ),
            (
                "Transition": "4→5",
                "Condition": "Кран 12 открылся И кран 9 закрылся И Pтг > 1.96",
                "AlgCondition": "[am.KR12.isON AND am.KR9.isOff AND aipar.Ptg_inTRK.value > 1.96]"
            ),
            (
                "Step": "5",
                "Commands": [
                    (
                        "Command": "Закрытие крана 12, открытие крана 9",
                        "AlgCommand": "[cmd_KR12_Off]",
                        "Fault": "Кран 12 не закрылся, кран 9 не открылся",
                        "AlgFault": "[am.KR12.notOff OR am.KR9.notOn]"
                    )
                ]
            ),
            (
                "Transition": "5→6",
                "Condition": "Кран 12 закрылся И кран 9 открылся",
                "AlgCondition": "[am.KR12.isOFF AND am.KR9.isON]"
            ),
            (
                "Step": "6",
                "Commands": [
                    (
                        "Command": "Кран 6 закрыть",
                        "AlgCommand": "[cmd_Kr6_Off]",
                        "Fault": "Кран 6 не закрылся",
                        "AlgFault": "[am.Kr6.notOff]"
                    )
                ]
            ),
            (
                "Transition": "6→7",
                "Condition": "Кран 6 закрыт",
                "AlgCondition": "[am.Kr6.isOFF]"
            ),
            (
                "Step": "7",
                "Commands": [
                    (
                        "Command": "Кран 1 закрыть",
                        "AlgCommand": "[cmd_Kr1_Off]",
                        "Fault": "Кран 1 не закрылся",
                        "AlgFault": "[am.Kr1.notOff]"
                    ),
                    (
                        "Command": "Кран 2 закрыть",
                        "AlgCommand": "[cmd_Kr2_Off]",
                        "Fault": "Кран 2 не закрылся",
                        "AlgFault": "[am.Kr2.notOff]"
                    ),
                    (
                        "Command": "Кран 4 открыть",
                        "AlgCommand": "[cmd_Kr4_On]",
                        "Fault": "Кран 4 не открылся",
                        "AlgFault": "[am.Kr4.notOn]"
                    )
                ]
            ),
            (
                "Transition": "7→8",
                "Condition": "Кран 1 закрыт И Кран 2 закрыт И Кран 4 открыт",
                "AlgCondition": "[am.Kr1.isOFF AND am.Kr2.isOFF AND am.Kr4.isON]"
            ),
            (
                "Step": "8",
                "Commands": [
                    (
                        "Command": "Завершение",
                        "AlgCommand": "[finish]"
                    )
                ]
            ),
            (
                "Transition": "8→0",
                "Condition": "Логическая 1",
                "AlgCondition": "[TRUE]"
            ),
            (
                "Transition": "N→0",
                "Condition": "Снятие режима",
                "AlgCondition": "[NOT mde.KPK]"
            )
        ]
    )
)'}
	KPK : T_KPK; //КПК
{attribute 'export' := '(
    "type": "TSequence",
    "sequence": (
        "Group": "Режимные",
        "AlgGroup": "smd",
        "Name": "АПК",
        "Alg": "[APK]",
        "Items": [
            (
                "Transition": "0→1",
                "Condition": "Режим АПК",
                "AlgCondition": "[mde.APK]"
            ),
            (
                "Step": "1",
                "Commands": [
                    (
                        "Command": "Предпусковая сигнализация",
                        "AlgCommand": "[cmd_sound_On]"
                    )
                ]
            ),
            (
                "Transition": "1→2",
                "Condition": "Логическая 1",
                "AlgCondition": "[TRUE]",
                "DelayTime": "10"
            ),
            (
                "Step": "2",
                "Commands": [
                    (
                        "Command": "Включение маслонасосов смазки и уплотнения",
                        "AlgCommand": "[cmd_PNU_S_On]"
                    )
                ]
            ),
            (
                "Transition": "2→3",
                "Condition": "dP масло-газ > 0.5 кгс/см2 и Pm > 1 кгс/см2",
                "AlgCondition": "[aipar.dPmg.value > 0.5 AND NOT dipar.Pm_N_Pn.value]"
            ),
            (
                "Step": "3",
                "Commands": [
                    (
                        "Command": "Взвод защиты по маслосистеме нагнетателя",
                        "AlgCommand": "[cmd_shPmN_On]"
                    ),
                    (
                        "Command": "Взвод защиты по перепаду \"масло-газ\"",
                        "AlgCommand": "[cmd_sh_dPmg_On]"
                    ),
                    (
                        "Command": "Запуск последовательности \"Заполнение контура компрессора\"",
                        "AlgCommand": "[cmd_filling]",
                        "Classifier": "P"
                    )
                ]
            ),
            (
                "Transition": "3→4",
                "Condition": "Подсистема \"Газовая обвязка\" запущена",
                "AlgCondition": "[Filling.finish]"
            ),
            (
                "Step": "4",
                "Commands": [
                    (
                        "Command": "Запуск последовательности \"Пуск двигателя\"",
                        "AlgCommand": "[cmd_start_D]",
                        "Classifier": "P"
                    )
                ]
            ),
            (
                "Transition": "4→5",
                "Condition": "Двигатель перешел в режим \"Работа\"",
                "AlgCondition": "[FuelReg.fReg.started]",
                "DelayTime": "*"
            ),
            (
                "Step": "5",
                "Commands": [
                    (
                        "Command": "Завершение",
                        "AlgCommand": "[finish]"
                    )
                ]
            ),
            (
                "Transition": "5→0",
                "Condition": "Логическая 1",
                "AlgCondition": "[TRUE]"
            ),
            (
                "Transition": "N→0",
                "Condition": "Режимы аварийного останова",
                "AlgCondition": "[alg.AO]"
            )
        ]
    )
)'}
	APK : T_APK; //АПК
{attribute 'export' := '(
    "type": "TSequence",
    "sequence": (
        "Group": "Режимные",
        "AlgGroup": "smd",
        "Name": "Переход К-М",
        "Alg": "[K_M]",
        "Items": [
            (
                "Transition": "0→1",
                "Condition": "(Режим Переход К-М)",
                "AlgCondition": "[mde.K_M]"
            ),
            (
                "Step": "1",
                "Commands": [
                    (
                        "Command": "Кран 2 открыть",
                        "AlgCommand": "[cmd_Kr2_On]",
                        "Fault": "Кран 2 не открылся",
                        "AlgFault": "[am.Kr2.notOn]"
                    )
                ]
            ),
            (
                "Transition": "1→2",
                "Condition": "Кран 2 открыт",
                "AlgCondition": "[am.Kr2.isON]"
            ),
            (
                "Step": "2",
                "Commands": [
                    (
                        "Command": "Кран 6 закрыть",
                        "AlgCommand": "[cmd_Kr6_Off]",
                        "Fault": "Кран 6 не закрылся",
                        "AlgFault": "[am.Kr6.notOff]"
                    )
                ]
            ),
            (
                "Transition": "2→3",
                "Condition": "Кран 6 закрыт",
                "AlgCondition": "[am.Kr6.isOff]"
            ),
            (
                "Step": "3",
                "Commands": [
                    (
                        "Command": "Завершение",
                        "AlgCommand": "[finish]"
                    )
                ]
            ),
            (
                "Transition": "3→0",
                "Condition": "Логическая 1",
                "AlgCondition": "[TRUE]"
            ),
            (
                "Transition": "N→0",
                "Condition": "Режимы аварийного останова ИЛИ Режим \"Переход М-К\"",
                "AlgCondition": "[alg.AO OR mde.M_K]"
            )
        ]
    )
)'}
	K_M : T_K_M; //Переход К-М
{attribute 'export' := '(
    "type": "TSequence",
    "sequence": (
        "Group": "Режимные",
        "AlgGroup": "smd",
        "Name": "Переход М-К",
        "Alg": "[M_K]",
        "Items": [
            (
                "Transition": "0→1",
                "Condition": "(Режим Переход М-К) ИЛИ (НОсс => Переход М-К) ИЛИ (НОбс => Переход М-К)",
                "AlgCondition": "[mde.M_K OR NOss.cmd_M_K OR NObs.cmd_M_K]"
            ),
            (
                "Step": "1",
                "Commands": [
                    (
                        "Command": "Кран 6 открыть",
                        "AlgCommand": "[cmd_KR6_On]",
                        "Fault": "Кран 6 не открылся",
                        "AlgFault": "[am.KR6.notOn]"
                    )
                ]
            ),
            (
                "Transition": "1→2",
                "Condition": "Кран 6 открыт",
                "AlgCondition": "[am.Kr6.isON]"
            ),
            (
                "Step": "2",
                "Commands": [
                    (
                        "Command": "Кран 2 закрыть",
                        "AlgCommand": "[cmd_Kr2_Off]",
                        "Fault": "Кран 2 не закрылся",
                        "AlgFault": "[am.Kr2.notOff]"
                    )
                ]
            ),
            (
                "Transition": "2→3",
                "Condition": "Кран 2 закрыт",
                "AlgCondition": "[am.Kr2.isOFF]"
            ),
            (
                "Step": "3",
                "Commands": [
                    (
                        "Command": "Завершение",
                        "AlgCommand": "[finish]"
                    )
                ]
            ),
            (
                "Transition": "3→0",
                "Condition": "Логическая 1",
                "AlgCondition": "[TRUE]"
            ),
            (
                "Transition": "N→0",
                "Condition": "Режим АОсс ИЛИ Режим АОбс ИЛИ Режим \"Переход К-М\"",
                "AlgCondition": "[mde.AOss OR mde.AObs OR mde.K_M]"
            )
        ]
    )
)'}
	M_K : T_M_K; //Переход М-К
{attribute 'export' := '(
    "type": "TSequence",
    "sequence": (
        "Group": "Режимные",
        "AlgGroup": "smd",
        "Name": "НОсс",
        "Alg": "[NOss]",
        "Items": [
            (
                "Transition": "0→1",
                "Condition": "Режим НОсс",
                "AlgCondition": "[mde.NOss]"
            ),
            (
                "Step": "1",
                "Commands": [
                    (
                        "Command": "Запуск последовательности \"Переход М-К\"",
                        "AlgCommand": "[cmd_M_K]",
                        "Classifier": "P"
                    )
                ]
            ),
            (
                "Transition": "1→2",
                "Condition": "Последовательность \"Переход М-К\" завершена",
                "AlgCondition": "[M_K.finish]"
            ),
            (
                "Step": "2",
                "Commands": [
                    (
                        "Command": "Снятие защиты по маслосистеме ТК и СТ",
                        "AlgCommand": "[sh_ms_off]"
                    ),
                    (
                        "Command": "Нормальный останов двигателя",
                        "AlgCommand": "[alg.normalStopCom]",
                        "Fault": "Д не перешел на малый газ для охлаждения",
                        "AlgFault": "[NOT FuelReg.fReg.cooling]",
                        "Classifier": "S"
                    )
                ]
            ),
            (
                "Transition": "2→3",
                "Condition": "Двигатель перешел на малый газ для охлаждения",
                "AlgCondition": "[FuelReg.fReg.cooling]",
                "DelayTime": "10"
            ),
            (
                "Step": "3",
                "Commands": [
                    (
                        "Command": "Охлаждение двигателя",
                        "AlgCommand": "[cooling]"
                    )
                ]
            ),
            (
                "Transition": "3→4",
                "Condition": "Охлаждение двигателя завершено",
                "AlgCondition": "[NOT FuelReg.fReg.cooling]",
                "DelayTime": "*"
            ),
            (
                "Step": "4",
                "Commands": [
                    (
                        "Command": "Нормальный останов двигателя",
                        "AlgCommand": "[alg.normalStopCom]",
                        "Classifier": "R"
                    ),
                    (
                        "Command": "Включение маслонасосов смазки и уплотнения",
                        "AlgCommand": "[cmd_PNU_S_On]"
                    ),
                    (
                        "Command": "Включение Э/М ВНА",
                        "AlgCommand": "[cmd_VNA_On]",
                        "Classifier": "S"
                    ),
                    (
                        "Command": "Открыть КПВ 2, 3, 4",
                        "AlgCommand": "[cmd_KPV234_On]",
                        "Fault": "КПВ 2, 3, 4 не открылись",
                        "AlgFault": "[am.KPV2.notOn OR am.KPV3.notOn OR am.KPV4.notOn]"
                    ),
                    (
                        "Command": "Закрытие крана 12, открытие крана 9",
                        "AlgCommand": "[cmd_KR12_Off]",
                        "Fault": "Кран 12 не закрылся, кран 9 не открылся",
                        "AlgFault": "[am.KR12.notOff OR am.KR9.notOn]"
                    ),
                    (
                        "Command": "Снятие защиты по ТГ",
                        "AlgCommand": "[cmd_sh_TG_Off]"
                    ),
                    (
                        "Command": "СК закрыть",
                        "AlgCommand": "[cmd_SK_Off]"
                    )
                ]
            ),
            (
                "Transition": "4→5",
                "Condition": "Подача топливного газа прекращена",
                "AlgCondition": "[am.KR9.ison AND am.KR12.isOff]"
            ),
            (
                "Step": "5",
                "Commands": [
                    (
                        "Command": "Выбег нагнетателя",
                        "AlgCommand": "[check_Nst]"
                    )
                ]
            ),
            (
                "Transition": "5→6",
                "Condition": "Nст < 100 об/мин",
                "AlgCondition": "[acpar.Nst.value < 100.0]"
            ),
            (
                "Step": "6",
                "Commands": [
                    (
                        "Command": "Запуск последовательности \"Стравливание контура компрессора\"",
                        "AlgCommand": "[cmd_bleeding]",
                        "Classifier": "P"
                    )
                ]
            ),
            (
                "Transition": "6→7",
                "Condition": "Подрежим \"Стравливание контура компрессора\" завершен",
                "AlgCondition": "[bleeding.finish]"
            ),
            (
                "Step": "7",
                "Commands": [
                    (
                        "Command": "Снятие защиты по перепаду \"масло-газ\"",
                        "AlgCommand": "[cmd_sh_dPmg_Off]"
                    ),
                    (
                        "Command": "Пуск таймера отключения ПНС, ПНУ",
                        "AlgCommand": "[cmd_PNU_S_Off]",
                        "Classifier": "P"
                    ),
                    (
                        "Command": "Выбег двигателя",
                        "AlgCommand": "[check_Ntk]"
                    )
                ]
            ),
            (
                "Transition": "7→8",
                "Condition": "Nтк < 100 об/мин",
                "AlgCondition": "[acpar.Ntk.value < 100.0]",
                "DelayTime": "2"
            ),
            (
                "Step": "8",
                "Commands": [
                    (
                        "Command": "Отключение Э/М ВНА",
                        "AlgCommand": "[cmd_VNA_On]",
                        "Classifier": "R"
                    ),
                    (
                        "Command": "Снятие защиты по маслосистеме нагнетателя",
                        "AlgCommand": "[cmd_shPmN_Off]"
                    ),
                    (
                        "Command": "Пуск таймера отключения ПНС, ПНУ",
                        "AlgCommand": "[cmd_PNU_S_Off]",
                        "Classifier": "P"
                    ),
                    (
                        "Command": "Завершение",
                        "AlgCommand": "[finish]"
                    )
                ]
            ),
            (
                "Transition": "8→0",
                "Condition": "Логическая 1",
                "AlgCondition": "[TRUE]"
            ),
            (
                "Transition": "N→0",
                "Condition": "Режим АОсс",
                "AlgCondition": "[mde.AOss]"
            )
        ]
    )
)'}
	NOss : T_NOss; //НОсс
{attribute 'export' := '(
    "type": "TSequence",
    "sequence": (
        "Group": "Режимные",
        "AlgGroup": "smd",
        "Name": "НОбс",
        "Alg": "[NObs]",
        "Items": [
            (
                "Transition": "0→1",
                "Condition": "Режим НОбс",
                "AlgCondition": "[mde.NObs]"
            ),
            (
                "Step": "1",
                "Commands": [
                    (
                        "Command": "Запуск последовательности \"Переход М-К\"",
                        "AlgCommand": "[cmd_M_K]",
                        "Classifier": "P"
                    )
                ]
            ),
            (
                "Transition": "1→2",
                "Condition": "Последовательность \"Переход М-К\" завершена",
                "AlgCondition": "[M_K.finish]"
            ),
            (
                "Step": "2",
                "Commands": [
                    (
                        "Command": "Снятие защиты по маслосистеме ТК и СТ",
                        "AlgCommand": "[sh_ms_off]"
                    ),
                    (
                        "Command": "Нормальный останов двигателя",
                        "AlgCommand": "[alg.normalStopCom]",
                        "Fault": "Д не перешел на малый газ для охлаждения",
                        "AlgFault": "[NOT FuelReg.fReg.cooling]",
                        "Classifier": "S"
                    )
                ]
            ),
            (
                "Transition": "2→3",
                "Condition": "Двигатель перешел на малый газ для охлаждения",
                "AlgCondition": "[FuelReg.fReg.cooling]",
                "DelayTime": "10"
            ),
            (
                "Step": "3",
                "Commands": [
                    (
                        "Command": "Охлаждение двигателя",
                        "AlgCommand": "[cooling]"
                    )
                ]
            ),
            (
                "Transition": "3→4",
                "Condition": "Охлаждение двигателя завершено",
                "AlgCondition": "[NOT FuelReg.fReg.cooling]",
                "DelayTime": "*"
            ),
            (
                "Step": "4",
                "Commands": [
                    (
                        "Command": "Нормальный останов двигателя",
                        "AlgCommand": "[alg.normalStopCom]",
                        "Classifier": "R"
                    ),
                    (
                        "Command": "Включение маслонасосов смазки и уплотнения",
                        "AlgCommand": "[cmd_PNU_S_On]"
                    ),
                    (
                        "Command": "Включение Э/М ВНА",
                        "AlgCommand": "[cmd_VNA_On]",
                        "Classifier": "S"
                    ),
                    (
                        "Command": "Открыть КПВ 2, 3, 4",
                        "AlgCommand": "[cmd_KPV234_On]",
                        "Fault": "КПВ 2, 3, 4 не открылись",
                        "AlgFault": "[am.KPV2.notOn OR am.KPV3.notOn OR am.KPV4.notOn]"
                    ),
                    (
                        "Command": "Закрытие крана 12, открытие крана 9",
                        "AlgCommand": "[cmd_KR12_Off]",
                        "Fault": "Кран 12 не закрылся, кран 9 не открылся",
                        "AlgFault": "[am.KR12.notOff OR am.KR9.notOn]"
                    ),
                    (
                        "Command": "Снятие защиты по ТГ",
                        "AlgCommand": "[cmd_sh_TG_Off]"
                    ),
                    (
                        "Command": "СК закрыть",
                        "AlgCommand": "[cmd_SK_Off]"
                    )
                ]
            ),
            (
                "Transition": "4→5",
                "Condition": "Подача топливного газа прекращена",
                "AlgCondition": "[am.KR9.ison AND am.KR12.isOff]"
            ),
            (
                "Step": "5",
                "Commands": [
                    (
                        "Command": "Выбег нагнетателя",
                        "AlgCommand": "[check_Nst]"
                    )
                ]
            ),
            (
                "Transition": "5→6",
                "Condition": "Nст < 100 об/мин",
                "AlgCondition": "[acpar.Nst.value < 100.0]"
            ),
            (
                "Step": "6",
                "Commands": [
                    (
                        "Command": "Кран 1 закрыть",
                        "AlgCommand": "[cmd_Kr1_Off]",
                        "Fault": "Кран 1 не закрылся",
                        "AlgFault": "[am.Kr1.notOff]"
                    ),
                    (
                        "Command": "Кран 6 закрыть",
                        "AlgCommand": "[cmd_Kr6_Off]",
                        "Fault": "Кран 6 не закрылся",
                        "AlgFault": "[am.Kr6.notOff]"
                    ),
                    (
                        "Command": "Кран 4 открыть",
                        "AlgCommand": "[cmd_Kr4_On]",
                        "Fault": "Кран 4 не открылся",
                        "AlgFault": "[am.Kr4.notOn]"
                    )
                ]
            ),
            (
                "Transition": "6→7",
                "Condition": "Кран 1 закрыт И Кран 6 закрыт И Кран 4 открыт",
                "AlgCondition": "[am.Kr1.isOFF AND am.Kr6.isOFF AND am.Kr4.isON]"
            ),
            (
                "Step": "7",
                "Commands": [
                    (
                        "Command": "Выбег двигателя",
                        "AlgCommand": "[check_Ntk]"
                    )
                ]
            ),
            (
                "Transition": "7→8",
                "Condition": "Nтк < 100 об/мин",
                "AlgCondition": "[acpar.Ntk.value < 100.0]"
            ),
            (
                "Step": "8",
                "Commands": [
                    (
                        "Command": "Отключение Э/М ВНА",
                        "AlgCommand": "[cmd_VNA_On]",
                        "Classifier": "R"
                    ),
                    (
                        "Command": "Завершение",
                        "AlgCommand": "[finish]",
                        "Classifier": "P"
                    )
                ]
            ),
            (
                "Transition": "8→0",
                "Condition": "Логическая 1",
                "AlgCondition": "[TRUE]"
            ),
            (
                "Transition": "N→0",
                "Condition": "Режим АОбс",
                "AlgCondition": "[mde.AObs]"
            )
        ]
    )
)'}
	NObs : T_NObs; //НОбс
{attribute 'export' := '(
    "type": "TSequence",
    "sequence": (
        "Group": "Режимные",
        "AlgGroup": "smd",
        "Name": "АОсс",
        "Alg": "[AOss]",
        "Items": [
            (
                "Transition": "0→1",
                "Condition": "Режим АОсс",
                "AlgCondition": "[mde.AOss]"
            ),
            (
                "Step": "1",
                "Commands": [
                    (
                        "Command": "Аварийный останов двигателя",
                        "AlgCommand": "[emergStopCom]",
                        "Classifier": "S"
                    ),
                    (
                        "Command": "Запуск последовательности \"Переход М-К\"",
                        "AlgCommand": "[cmd_M_K]",
                        "Classifier": "P"
                    ),
                    (
                        "Command": "Снятие защиты по маслосистеме ТК и СТ",
                        "AlgCommand": "[sh_ms_off]"
                    ),
                    (
                        "Command": "Открыть КПВ 1, 5",
                        "AlgCommand": "[cmd_KPV15_On]",
                        "Fault": "КПВ 1, 5 не открылись",
                        "AlgFault": "[am.KPV1.notOn AND am.KPV5.notOn]"
                    ),
                    (
                        "Command": "Открыть КПВ 2, 3, 4",
                        "AlgCommand": "[cmd_KPV234_On]",
                        "Fault": "КПВ 2, 3, 4 не открылись",
                        "AlgFault": "[am.KPV2.notOn OR am.KPV3.notOn OR am.KPV4.notOn]"
                    ),
                    (
                        "Command": "Включение Э/М ВНА",
                        "AlgCommand": "[cmd_VNA_On]",
                        "Classifier": "S"
                    ),
                    (
                        "Command": "Снятие защиты по ТГ",
                        "AlgCommand": "[cmd_sh_TG_Off]"
                    ),
                    (
                        "Command": "Включение маслонасосов смазки и уплотнения",
                        "AlgCommand": "[cmd_PNU_S_On]"
                    ),
                    (
                        "Command": "Закрытие крана 12, открытие крана 9",
                        "AlgCommand": "[cmd_KR12_Off]",
                        "Fault": "Кран 12 не закрылся, кран 9 не открылся",
                        "AlgFault": "[am.KR12.notOff OR am.KR9.notOn]"
                    ),
                    (
                        "Command": "Останов воздушного стартера",
                        "AlgCommand": "[cmd_VS_Off]",
                        "Fault": "Кран 13 не закрылся",
                        "AlgFault": "[am.KR13.notOff]"
                    ),
                    (
                        "Command": "Кран 15 закрыть",
                        "AlgCommand": "[am.KR15.on]",
                        "Fault": "Кран 15 не закрылся",
                        "AlgFault": "[am.KR15.notOff]",
                        "Classifier": "R"
                    ),
                    (
                        "Command": "Кран 4 закрыть",
                        "AlgCommand": "[cmd_Kr4_Off]",
                        "Fault": "Кран 4 не закрылся",
                        "AlgFault": "[am.Kr4.notOff]"
                    ),
                    (
                        "Command": "Закрытие крана 11, открытие крана 10",
                        "AlgCommand": "[cmd_KR11_Off]"
                    ),
                    (
                        "Command": "Проверка Nст",
                        "AlgCommand": "[check_Nst]",
                        "Fault": "Nст > 100 об/мин",
                        "AlgFault": "[acpar.Nst.value > 100.0]"
                    )
                ]
            ),
            (
                "Transition": "1→2",
                "Condition": "Кран 4 закрыт И Nст < 100 об/мин",
                "AlgCondition": "[am.Kr4.isOFF AND ( acpar.Nst.value < 100.0 OR acpar.Nst.flt )]",
                "DelayTime": "10"
            ),
            (
                "Step": "2",
                "Commands": [
                    (
                        "Command": "Запуск последовательности \"Стравливание контура компрессора\"",
                        "AlgCommand": "[cmd_bleeding]",
                        "Classifier": "P"
                    )
                ]
            ),
            (
                "Transition": "2→3",
                "Condition": "Подрежим \"Стравливание контура компрессора\" завершен",
                "AlgCondition": "[bleeding.finish]"
            ),
            (
                "Step": "3",
                "Commands": [
                    (
                        "Command": "Выбег двигателя",
                        "AlgCommand": "[check_Ntk]"
                    )
                ]
            ),
            (
                "Transition": "3→4",
                "Condition": "Логическая 1",
                "AlgCondition": "[TRUE]",
                "DelayTime": "60"
            ),
            (
                "Step": "4",
                "Commands": [
                    (
                        "Command": "Отключение Э/М ВНА",
                        "AlgCommand": "[cmd_VNA_On]",
                        "Classifier": "R"
                    ),
                    (
                        "Command": "Снятие защиты по маслосистеме нагнетателя",
                        "AlgCommand": "[cmd_shPmN_Off]"
                    ),
                    (
                        "Command": "Снятие защиты по перепаду \"масло-газ\"",
                        "AlgCommand": "[cmd_sh_dPmg_Off]"
                    )
                ]
            ),
            (
                "Transition": "4→5",
                "Condition": "Логическая 1",
                "AlgCondition": "[TRUE]",
                "DelayTime": "2"
            ),
            (
                "Step": "5",
                "Commands": [
                    (
                        "Command": "Пуск таймера отключения ПНС, ПНУ",
                        "AlgCommand": "[cmd_PNU_S_Off]"
                    )
                ]
            ),
            (
                "Transition": "5→6",
                "Condition": "Логическая 1",
                "AlgCondition": "[TRUE]"
            ),
            (
                "Step": "6",
                "Commands": [
                    (
                        "Command": "Завершение",
                        "AlgCommand": "[finish]",
                        "Fault": "АОсс завершен, нажмите кнопку \"Деблокировка\"",
                        "AlgFault": "[NOT tch.Unlock.value]"
                    )
                ]
            ),
            (
                "Transition": "6→0",
                "Condition": "Деблокировка",
                "AlgCondition": "[tch.Unlock.value]"
            ),
            (
                "Transition": "N→0",
                "Condition": "Снятие режима",
                "AlgCondition": "[NOT mde.AOss]"
            )
        ]
    )
)'}
	AOss : T_AOss; //АОсс
{attribute 'export' := '(
    "type": "TSequence",
    "sequence": (
        "Group": "Режимные",
        "AlgGroup": "smd",
        "Name": "АОбс",
        "Alg": "[AObs]",
        "Items": [
            (
                "Transition": "0→1",
                "Condition": "Режим АОбс",
                "AlgCondition": "[mde.AObs]"
            ),
            (
                "Step": "1",
                "Commands": [
                    (
                        "Command": "Аварийный останов двигателя",
                        "AlgCommand": "[emergStopCom]",
                        "Classifier": "S"
                    ),
                    (
                        "Command": "Запуск последовательности \"Переход М-К\"",
                        "AlgCommand": "[cmd_M_K]",
                        "Classifier": "P"
                    ),
                    (
                        "Command": "Снятие защиты по маслосистеме ТК и СТ",
                        "AlgCommand": "[sh_ms_off]"
                    ),
                    (
                        "Command": "Открыть КПВ 1, 5",
                        "AlgCommand": "[cmd_KPV15_On]",
                        "Fault": "КПВ 1, 5 не открылись",
                        "AlgFault": "[am.KPV1.notOn AND am.KPV5.notOn]"
                    ),
                    (
                        "Command": "Открыть КПВ 2, 3, 4",
                        "AlgCommand": "[cmd_KPV234_On]",
                        "Fault": "КПВ 2, 3, 4 не открылись",
                        "AlgFault": "[am.KPV2.notOn OR am.KPV3.notOn OR am.KPV4.notOn]"
                    ),
                    (
                        "Command": "Включение Э/М ВНА",
                        "AlgCommand": "[cmd_VNA_On]",
                        "Classifier": "S"
                    ),
                    (
                        "Command": "Снятие защиты по ТГ",
                        "AlgCommand": "[cmd_sh_TG_Off]"
                    ),
                    (
                        "Command": "Включение маслонасосов смазки и уплотнения",
                        "AlgCommand": "[cmd_PNU_S_On]"
                    ),
                    (
                        "Command": "Закрытие крана 12, открытие крана 9",
                        "AlgCommand": "[cmd_KR12_Off]",
                        "Fault": "Кран 12 не закрылся, кран 9 не открылся",
                        "AlgFault": "[am.KR12.notOff OR am.KR9.notOn]"
                    ),
                    (
                        "Command": "Останов воздушного стартера",
                        "AlgCommand": "[cmd_VS_Off]",
                        "Fault": "Кран 13 не закрылся",
                        "AlgFault": "[am.KR13.notOff]"
                    ),
                    (
                        "Command": "Кран 15 закрыть",
                        "AlgCommand": "[am.KR15.on]",
                        "Fault": "Кран 15 не закрылся",
                        "AlgFault": "[am.KR15.notOff]",
                        "Classifier": "R"
                    ),
                    (
                        "Command": "Кран 4 закрыть",
                        "AlgCommand": "[cmd_Kr4_Off]",
                        "Fault": "Кран 4 не закрылся",
                        "AlgFault": "[am.Kr4.notOff]"
                    ),
                    (
                        "Command": "Закрытие крана 11, открытие крана 10",
                        "AlgCommand": "[cmd_KR11_Off]"
                    ),
                    (
                        "Command": "Проверка Nст",
                        "AlgCommand": "[check_Nst]",
                        "Fault": "Nст > 100 об/мин",
                        "AlgFault": "[acpar.Nst.value > 100.0]"
                    )
                ]
            ),
            (
                "Transition": "1→2",
                "Condition": "Кран 4 закрыт И Nст < 100 об/мин",
                "AlgCondition": "[am.Kr4.isOFF AND ( acpar.Nst.value < 100.0 OR acpar.Nst.flt )]",
                "DelayTime": "10"
            ),
            (
                "Step": "2",
                "Commands": [
                    (
                        "Command": "Выбег двигателя",
                        "AlgCommand": "[check_Ntk]"
                    )
                ]
            ),
            (
                "Transition": "2→3",
                "Condition": "Логическая 1",
                "AlgCondition": "[TRUE]",
                "DelayTime": "60"
            ),
            (
                "Step": "3",
                "Commands": [
                    (
                        "Command": "Отключение Э/М ВНА",
                        "AlgCommand": "[cmd_VNA_On]",
                        "Classifier": "R"
                    ),
                    (
                        "Command": "Кран 1 закрыть",
                        "AlgCommand": "[cmd_Kr1_Off]",
                        "Fault": "Кран 1 не закрылся",
                        "AlgFault": "[am.Kr1.notOff]"
                    ),
                    (
                        "Command": "Кран 2 закрыть",
                        "AlgCommand": "[cmd_Kr2_Off]",
                        "Fault": "Кран 2 не закрылся",
                        "AlgFault": "[am.Kr2.notOff]"
                    ),
                    (
                        "Command": "Кран 6 закрыть",
                        "AlgCommand": "[cmd_Kr6_Off]",
                        "Fault": "Кран 6 не закрылся",
                        "AlgFault": "[am.Kr6.notOff]"
                    ),
                    (
                        "Command": "Кран 4 открыть",
                        "AlgCommand": "[cmd_Kr4_On]",
                        "Fault": "Кран 4 не открылся",
                        "AlgFault": "[am.Kr4.notOn]"
                    )
                ]
            ),
            (
                "Transition": "3→4",
                "Condition": "Кран 1 закрыт И Кран 2 закрыт И Кран 6 закрыт И Кран 4 открыт",
                "AlgCondition": "[am.Kr1.isOFF AND am.Kr2.isOFF AND am.Kr6.isOFF AND am.Kr4.isON]"
            ),
            (
                "Step": "4",
                "Commands": [
                    (
                        "Command": "Завершение",
                        "AlgCommand": "[finish]",
                        "Fault": "АОбс завершен, нажмите кнопку \"Деблокировка\"",
                        "AlgFault": "[NOT tch.Unlock.value]"
                    )
                ]
            ),
            (
                "Transition": "4→0",
                "Condition": "Деблокировка",
                "AlgCondition": "[tch.Unlock.value]"
            ),
            (
                "Transition": "N→0",
                "Condition": "Снятие режима",
                "AlgCondition": "[NOT mde.AObs]"
            )
        ]
    )
)'}
	AObs : T_AObs; //АОбс
{attribute 'export' := '(
    "type": "TSequence",
    "sequence": (
        "Group": "Режимные",
        "AlgGroup": "smd",
        "Name": "Стравливание",
        "Alg": "[Bleeding_full]",
        "Items": [
            (
                "Transition": "0→1",
                "Condition": "Нажата кнопка \"Стравливание\"",
                "AlgCondition": "[btn.Bleeding.out]"
            ),
            (
                "Step": "1",
                "Commands": [
                    (
                        "Command": "Запуск последовательности \"Стравливание контура компрессора\"",
                        "AlgCommand": "[cmd_bleeding]",
                        "Classifier": "P"
                    )
                ]
            ),
            (
                "Transition": "1→2",
                "Condition": "Подрежим \"Стравливание контура компрессора\" завершен",
                "AlgCondition": "[bleeding.finish]"
            ),
            (
                "Step": "2",
                "Commands": [
                    (
                        "Command": "Снятие защиты по перепаду \"масло-газ\"",
                        "AlgCommand": "[cmd_sh_dPmg_Off]"
                    ),
                    (
                        "Command": "Снятие защиты по маслосистеме нагнетателя",
                        "AlgCommand": "[cmd_shPmN_Off]"
                    ),
                    (
                        "Command": "Пуск таймера отключения ПНС, ПНУ",
                        "AlgCommand": "[cmd_PNU_S_Off]"
                    )
                ]
            ),
            (
                "Transition": "2→3",
                "Condition": "Логическая 1",
                "AlgCondition": "[TRUE]"
            ),
            (
                "Step": "3",
                "Commands": [
                    (
                        "Command": "Завершение",
                        "AlgCommand": "[finish]"
                    )
                ]
            ),
            (
                "Transition": "3→0",
                "Condition": "Логическая 1",
                "AlgCondition": "[TRUE]"
            ),
            (
                "Transition": "N→0",
                "Condition": "Режим АОсс",
                "AlgCondition": "[mde.AOss]"
            )
        ]
    )
)'}
	Bleeding_full : T_Bleeding_full; //Стравливание
{attribute 'export' := '(
    "type": "TSequence",
    "sequence": (
        "Group": "Режимные",
        "AlgGroup": "smd",
        "Name": "Контроль САУ",
        "Alg": "[Check_SAU]",
        "Items": [
            (
                "Transition": "0→1",
                "Condition": "Нажата одна из пусковых кнопок ИЛИ Кнопка \"Контроль САУ\" ИЛИ Каждые 12 часов",
                "AlgCondition": "[check.btn OR btn.Check_SAU.out OR check.tmr12H.Q]"
            ),
            (
                "Step": "1",
                "Commands": [
                    (
                        "Command": "Контроль виброаппаратуры двигателя",
                        "AlgCommand": "[cmd_check_VibD]"
                    ),
                    (
                        "Command": "Контроль БЗА двигателя",
                        "AlgCommand": "[cmd_check_BZA]"
                    ),
                    (
                        "Command": "Ожидание аварийных сигнализаций",
                        "AlgCommand": "[wait_crs]"
                    )
                ]
            ),
            (
                "Transition": "1→2",
                "Condition": "Сформированы аварийные сигнализации двигателя",
                "AlgCondition": "[crs.Vs_D_Av.signalization AND crs.BZA_alr.signalization AND crs.Vsst_HH.signalization AND crs.Vstk_HH.signalization]",
                "DelayTime": "10"
            ),
            (
                "Step": "2",
                "Commands": [
                    (
                        "Command": "Завершение",
                        "AlgCommand": "[finish]"
                    )
                ]
            ),
            (
                "Transition": "2→0",
                "Condition": "Логическая 1",
                "AlgCondition": "[TRUE]"
            ),
            (
                "Transition": "N→0",
                "Condition": "Деблокировка",
                "AlgCondition": "[btn.Cancel.out]"
            )
        ]
    )
)'}
	Check_SAU : T_Check_SAU; //Контроль САУ
{attribute 'export' := '(
    "type": "TSequence",
    "sequence": (
        "Group": "Режимные",
        "AlgGroup": "smd",
        "Name": "Комплексное тестирование",
        "Alg": "[testing]",
        "Items": [
            (
                "Transition": "0→1",
                "Condition": "Кнопка \"Комплексное тестирование включить\"",
                "AlgCondition": "[btn.test_on.out]"
            ),
            (
                "Step": "1",
                "Commands": [
                    (
                        "Command": "Переинициализирование переменных",
                        "AlgCommand": "[init]",
                        "Classifier": "P"
                    )
                ]
            ),
            (
                "Transition": "1→2",
                "Condition": "Логическая 1",
                "AlgCondition": "[TRUE]",
                "DelayTime": "10"
            ),
            (
                "Step": "2",
                "Commands": [
                    (
                        "Command": "Шаг проверки: ХП из ГР // Кнопка \"ГР\"",
                        "AlgCommand": "[btn.GR.cmd]",
                        "Classifier": "P"
                    )
                ]
            ),
            (
                "Transition": "2→3",
                "Condition": "Режим ГР",
                "AlgCondition": "[mde.GR]",
                "DelayTime": "10"
            ),
            (
                "Step": "3",
                "Commands": [
                    (
                        "Command": "Шаг проверки: ХП из ГР // Кнопка \"ХП\"",
                        "AlgCommand": "[btn.HP.cmd]",
                        "Classifier": "P"
                    )
                ]
            ),
            (
                "Transition": "3→4",
                "Condition": "Разрешение кнопки \"Пуск\"",
                "AlgCondition": "[btn.start.prm]"
            ),
            (
                "Step": "4",
                "Commands": [
                    (
                        "Command": "Шаг проверки: ХП из ГР // Кнопка \"Пуск\"",
                        "AlgCommand": "[btn.Start.cmd]",
                        "Classifier": "P"
                    )
                ]
            ),
            (
                "Transition": "4→5",
                "Condition": "Последовательность \"ХП\" завершена",
                "AlgCondition": "[HP.finish]"
            ),
            (
                "Step": "5",
                "Commands": [
                    (
                        "Command": "Шаг проверки: КПК из ГР // Кнопка \"КПК\"",
                        "AlgCommand": "[btn.KPK.cmd]",
                        "Classifier": "P"
                    )
                ]
            ),
            (
                "Transition": "5→6",
                "Condition": "Разрешение кнопки \"Пуск\"",
                "AlgCondition": "[btn.start.prm]"
            ),
            (
                "Step": "6",
                "Commands": [
                    (
                        "Command": "Шаг проверки: КПК из ГР // Кнопка \"Пуск\"",
                        "AlgCommand": "[btn.Start.cmd]",
                        "Classifier": "P"
                    )
                ]
            ),
            (
                "Transition": "6→7",
                "Condition": "Последовательность \"КПК\" завершена",
                "AlgCondition": "[KPK.finish]"
            ),
            (
                "Step": "7",
                "Commands": [
                    (
                        "Command": "Шаг проверки: АПК из ГР под газом // Кнопка \"АПК\"",
                        "AlgCommand": "[btn.APK.cmd]",
                        "Classifier": "P"
                    )
                ]
            ),
            (
                "Transition": "7→8",
                "Condition": "Разрешение кнопки \"Пуск\"",
                "AlgCondition": "[btn.start.prm]"
            ),
            (
                "Step": "8",
                "Commands": [
                    (
                        "Command": "Шаг проверки: АПК из ГР под газом // Кнопка \"Пуск\"",
                        "AlgCommand": "[btn.Start.cmd]",
                        "Classifier": "P"
                    )
                ]
            ),
            (
                "Transition": "8→9",
                "Condition": "Последовательность \"АПК\" завершена",
                "AlgCondition": "[APK.finish]"
            ),
            (
                "Step": "9",
                "Commands": [
                    (
                        "Command": "Шаг проверки: АОсс из Кольца // Кнопка \"АОсс\"",
                        "AlgCommand": "[btn.AOss.cmd]",
                        "Classifier": "P"
                    )
                ]
            ),
            (
                "Transition": "9→10",
                "Condition": "Последовательность \"АОсс\" завершена",
                "AlgCondition": "[AOss.finish]"
            ),
            (
                "Step": "10",
                "Commands": [
                    (
                        "Command": "Шаг проверки: АОсс из Кольца // Кнопка \"Деблокировка\"",
                        "AlgCommand": "[btn.Unlock.cmd]",
                        "Classifier": "P"
                    )
                ]
            ),
            (
                "Transition": "10→11",
                "Condition": "Режим Ремонт",
                "AlgCondition": "[mde.Repair]",
                "DelayTime": "10"
            ),
            (
                "Step": "11",
                "Commands": [
                    (
                        "Command": "Шаг проверки: АПК из ГР без газа // Кнопка \"ГР\"",
                        "AlgCommand": "[btn.GR.cmd]",
                        "Classifier": "P"
                    )
                ]
            ),
            (
                "Transition": "11→12",
                "Condition": "Режим ГР",
                "AlgCondition": "[mde.GR]",
                "DelayTime": "10"
            ),
            (
                "Step": "12",
                "Commands": [
                    (
                        "Command": "Шаг проверки: АПК из ГР без газа // Кнопка \"АПК\"",
                        "AlgCommand": "[btn.APK.cmd]",
                        "Classifier": "P"
                    )
                ]
            ),
            (
                "Transition": "12→13",
                "Condition": "Разрешение кнопки \"Пуск\"",
                "AlgCondition": "[btn.start.prm]"
            ),
            (
                "Step": "13",
                "Commands": [
                    (
                        "Command": "Шаг проверки: АПК из ГР без газа // Кнопка \"Пуск\"",
                        "AlgCommand": "[btn.Start.cmd]",
                        "Classifier": "P"
                    )
                ]
            ),
            (
                "Transition": "13→14",
                "Condition": "Последовательность \"АПК\" завершена",
                "AlgCondition": "[APK.finish]"
            ),
            (
                "Step": "14",
                "Commands": [
                    (
                        "Command": "Шаг проверки: НОсс из Кольца // Кнопка \"НОсс\"",
                        "AlgCommand": "[btn.NOss.cmd]",
                        "Classifier": "P"
                    )
                ]
            ),
            (
                "Transition": "14→15",
                "Condition": "Последовательность \"НОсс\" завершена",
                "AlgCondition": "[NOss.finish]"
            ),
            (
                "Step": "15",
                "Commands": [
                    (
                        "Command": "Шаг проверки: АПМ из ГР без газа // Кнопка \"ГР\"",
                        "AlgCommand": "[btn.GR.cmd]",
                        "Classifier": "P"
                    )
                ]
            ),
            (
                "Transition": "15→16",
                "Condition": "Режим ГР",
                "AlgCondition": "[mde.GR]",
                "DelayTime": "10"
            ),
            (
                "Step": "16",
                "Commands": [
                    (
                        "Command": "Шаг проверки: АОбс из Магистрали // Кнопка \"АОбс\"",
                        "AlgCommand": "[btn.AObs.cmd]",
                        "Classifier": "P"
                    )
                ]
            ),
            (
                "Transition": "16→17",
                "Condition": "Последовательность \"АОбс\" завершена",
                "AlgCondition": "[AObs.finish]"
            ),
            (
                "Step": "17",
                "Commands": [
                    (
                        "Command": "Шаг проверки: АОбс из Магистрали // Кнопка \"Деблокировка\"",
                        "AlgCommand": "[btn.Unlock.cmd]",
                        "Classifier": "P"
                    )
                ]
            ),
            (
                "Transition": "17→18",
                "Condition": "Режим Ремонт",
                "AlgCondition": "[mde.Repair]",
                "DelayTime": "10"
            ),
            (
                "Step": "18",
                "Commands": [
                    (
                        "Command": "Шаг проверки: Переход М-К // Кнопка \"Переход М-К\"",
                        "AlgCommand": "[btn.M_K.cmd]",
                        "Classifier": "P"
                    )
                ]
            ),
            (
                "Transition": "18→19",
                "Condition": "Последовательность \"Переход М-К\" завершена",
                "AlgCondition": "[M_K.finish]"
            ),
            (
                "Step": "19",
                "Commands": [
                    (
                        "Command": "Шаг проверки: Повышение Nст до 5000 об/мин",
                        "AlgCommand": "[cmd_Nst_5000]",
                        "Fault": "Nст < 5000 об/мин",
                        "AlgFault": "[acpar.Nst.value < 5000]",
                        "Classifier": "P"
                    )
                ]
            ),
            (
                "Transition": "19→20",
                "Condition": "Nст > 4990 об/мин",
                "AlgCondition": "[acpar.Nst.value > 4990]"
            ),
            (
                "Step": "20",
                "Commands": [
                    (
                        "Command": "Шаг проверки: Переход К-М // Кнопка \"Переход К-М\"",
                        "AlgCommand": "[btn.K_M.cmd]",
                        "Classifier": "P"
                    )
                ]
            ),
            (
                "Transition": "20→21",
                "Condition": "Последовательность \"Переход К-М\" завершена",
                "AlgCondition": "[K_M.finish]"
            ),
            (
                "Step": "21",
                "Commands": [
                    (
                        "Command": "Шаг проверки: АОбс из Магистрали // Кнопка \"НОбс\"",
                        "AlgCommand": "[btn.NObs.cmd]",
                        "Classifier": "P"
                    )
                ]
            ),
            (
                "Transition": "21→22",
                "Condition": "Последовательность \"НОбс\" завершена",
                "AlgCondition": "[NObs.finish]"
            ),
            (
                "Step": "22",
                "Commands": [
                    (
                        "Command": "Шаг проверки: Стравливание из ГР под газом // Кнопка \"Стравливание ЦБК\"",
                        "AlgCommand": "[btn.Bleeding.cmd]"
                    )
                ]
            ),
            (
                "Transition": "22→23",
                "Condition": "Последовательность \"Стравливание\" завершена",
                "AlgCondition": "[Bleeding_full.finish]"
            ),
            (
                "Step": "23",
                "Commands": [
                    (
                        "Command": "Шаг проверки: Переход в Ремонт // Кнопка \"Ремонт\"",
                        "AlgCommand": "[btn.Repair.cmd]",
                        "Classifier": "P"
                    )
                ]
            ),
            (
                "Transition": "23→24",
                "Condition": "Режим Ремонт",
                "AlgCondition": "[mde.Repair]",
                "DelayTime": "10"
            ),
            (
                "Step": "24",
                "Commands": [
                    (
                        "Command": "Завершение",
                        "AlgCommand": "[finish]",
                        "Fault": "Нажмите кнопку \"Комплексное тестирование отключить\"",
                        "AlgFault": "[NOT btn.test_off.out]"
